// TIA Portal V20 export
DATA_BLOCK "IDB_LineD1"   // DB11
// stored: InstanceOfName LineD1.FB_LineD1, InstanceOfType FB, Namespace LineD1
"LineD1.FB_LineD1"
   // VAR
   //    "Conveyor_D1.1.1" : "Global.FB_Conveyor";
   //    "MABS_D1.1.1" : "Global.FB_MABS";
   //    "Transfer_D1.1.1" : "Global.FB_S300_tTransMode";
   // END_VAR
BEGIN
END_DATA_BLOCK
